Fanuc KAREL source: ka00195.KL

-- PROVISIONAL review KL for V770-1; original PC SHA256 8dbc40d85e4a854e0f4c2711655672d82e31a1420c635774c02aa4e773e04ff7
-- Incomplete behavior may be omitted. Consult companion uncertainty JSON. Do not deploy.
PROGRAM KA00195
%NOLOCKGROUP
-- UNRESOLVED_DECL SRC type=002017
-- UNRESOLVED_DECL DST type=002017
BEGIN
  -- UNRESOLVED_PC offsets 5-19; opcodes 22,22,1E
  -- UNRESOLVED_PC offsets 24-28; opcodes 7F
END KA00195
